TYPE ST_AllocationInfo:
STRUCT
		AllocationData 	:ARRAY[0..40] OF st_AllocationData;
END_STRUCT
END_TYPE

(* stored: Version 1.1.0.1, ProductVersion 3.1.4024.13
   DUT ST_AllocationInfo: Id {8384cd34-e95f-4efe-84d0-1d739ccbf987} *)
